// SIMATIC S7-200 project (STEP 7-Micro/WIN), CPU 221 REL 01.10

SYMBOL_TABLE USER1
wOpenRateFb1     VW0      // 开度反馈1
wOpenRateFb2     VW2      // 开度反馈2
wOpenRateRf1     VW4      // 开度设置1
wOpenRateRf2     VW6      // 开度设置2
dActionCount1    VD8      // 动作计数1
dActionCount2    VD12     // 动作计数2
aiOpenRateFb1    AIW0     // 开度反馈输入1
aiOpenRateFb2    AIW2     // 开度反馈输入2
aqOpenRateRf1    AQW2     // 开度设置输出1
aqOpenRateRf2    AQW4     // 开度设置输出2
END_SYMBOL_TABLE

ORGANIZATION_BLOCK MAIN:OB1
TITLE=PROGRAM COMMENTS
BEGIN
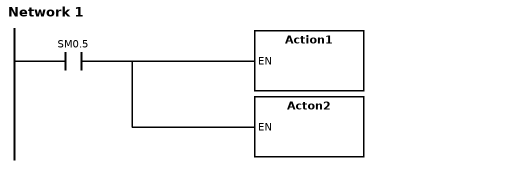
Network 1
LD     SM0.5
CALL   Action1:SBR0
CALL   Acton2:SBR1
END_ORGANIZATION_BLOCK

SUBROUTINE_BLOCK Action1:SBR0
TITLE=SUBROUTINE COMMENTS
BEGIN
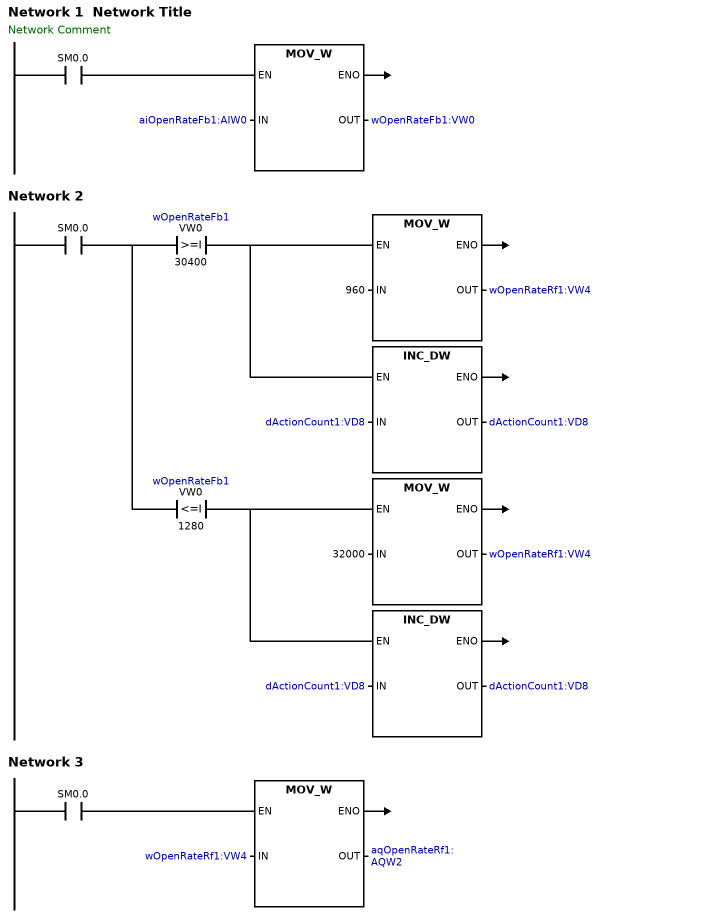
Network 1 // Network Title
// Network Comment
LD     SM0.0
MOVW   aiOpenRateFb1:AIW0, wOpenRateFb1:VW0
Network 2
LD     SM0.0
LPS
AW>=   wOpenRateFb1:VW0, 30400
MOVW   960, wOpenRateRf1:VW4
INCD   dActionCount1:VD8
LPP
AW<=   wOpenRateFb1:VW0, 1280
MOVW   32000, wOpenRateRf1:VW4
INCD   dActionCount1:VD8
Network 3
LD     SM0.0
MOVW   wOpenRateRf1:VW4, aqOpenRateRf1:AQW2
END_SUBROUTINE_BLOCK

SUBROUTINE_BLOCK Acton2:SBR1
TITLE=SUBROUTINE COMMENTS
BEGIN
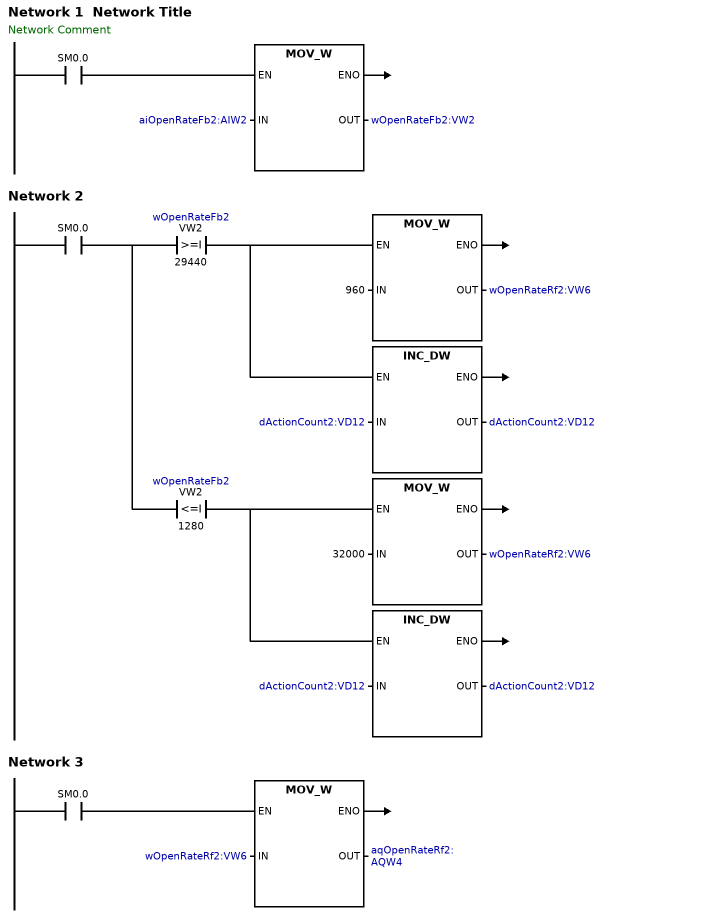
Network 1 // Network Title
// Network Comment
LD     SM0.0
MOVW   aiOpenRateFb2:AIW2, wOpenRateFb2:VW2
Network 2
LD     SM0.0
LPS
AW>=   wOpenRateFb2:VW2, 29440
MOVW   960, wOpenRateRf2:VW6
INCD   dActionCount2:VD12
LPP
AW<=   wOpenRateFb2:VW2, 1280
MOVW   32000, wOpenRateRf2:VW6
INCD   dActionCount2:VD12
Network 3
LD     SM0.0
MOVW   wOpenRateRf2:VW6, aqOpenRateRf2:AQW4
END_SUBROUTINE_BLOCK
